Staubli VAL3: getTool.pgx

public program getTool(tool& x_tTool[], num x_nIndex)
begin
  //
  x_tTool=saveTool:gun[x_nIndex]
end
